TYPE ST_KNXnetIP_ConnectionStateResponse EXTENDS ST_KNXnetIP_CommonHeader :
STRUCT
	nCommunicationChannelID		: BYTE;
	nStatusCode					: E_KNXnetIP_CONNECTIONSTATE_RESPONSE_ERROR;
END_STRUCT
END_TYPE

(* stored: Version 1.1.0.1
   DUT ST_KNXnetIP_ConnectionStateResponse: Id {82bfc511-bac8-454f-a418-1d0cde8d2259} *)
